(* task info with times of current task converted to millisecs and microsecs *)
FUNCTION_BLOCK FB_TaskTime
VAR_INPUT
END_VAR
VAR_OUTPUT
	bFirstCycle			: BOOL;		(* TRUE = 1st cycle of current task *)
	tTaskTimeMillisecs	: TIME;		(* Task Time in time format with ms resolution *)
	fTaskTimeMicrosecs	: LREAL;	(* Task Time in LREAL format with us resolution *)
	nTaskIndex			: BYTE;		(* Task Index of task where this FB is called *)
	nPLCPort			: UINT;		(* PLC port no *)
END_VAR
VAR
	fbTaskIndex			: GETCURTASKINDEX;
END_VAR
(*
-------------------------------------------------------------------------------------------------
Date		Version	Author	Comments
-------------------------------------------------------------------------------------------------
30/01/2015	3.00.00	PB		No change

-------------------------------------------------------------------------------------------------
15/03/2010	1.01.00	PB		Current PLC Port No added to FB_TaskTime
							bFirstCycle made primary output of FB_TaskTime
05/02/2010	1.00.00	PB		Initial release
							
-------------------------------------------------------------------------------------------------
*)

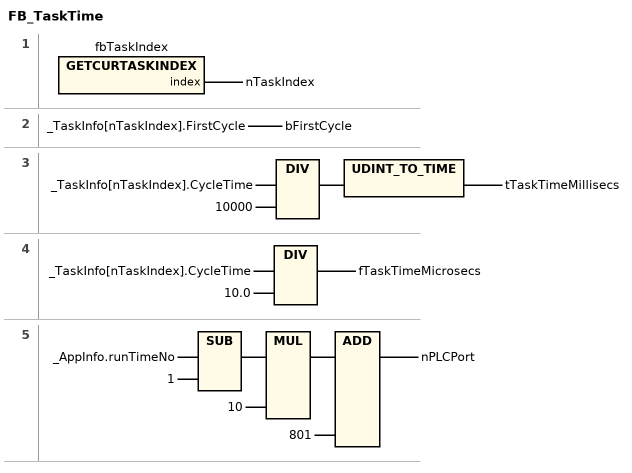
// NETWORK 1
fbTaskIndex(); // GETCURTASKINDEX
nTaskIndex := fbTaskIndex.index;

// NETWORK 2
bFirstCycle := _TaskInfo[nTaskIndex].FirstCycle;

// NETWORK 3
tTaskTimeMillisecs := UDINT_TO_TIME(_TaskInfo[nTaskIndex].CycleTime / 10000);

// NETWORK 4
fTaskTimeMicrosecs := _TaskInfo[nTaskIndex].CycleTime / 10.0;

// NETWORK 5
nPLCPort := (_AppInfo.runTimeNo - 1) * 10 + 801;

END_FUNCTION_BLOCK

(* stored: Version 1.1.0.1, ProductVersion 3.1.4024.15
   POU FB_TaskTime: Id {8bb5977a-ea81-4f29-8fbf-b5e65e44b3bd}, SpecialFunc None *)
